(* Logix 5000 project; controller cal1632 1756-L62 rev 16.20; software revision 16.05; part 60 of 61 *)
(* tags used below, declared in another part *)
   A02 : ALIAS FOR hmi_dint[0].2;
   A08 : ALIAS FOR hmi_dint[0].8;
   A09 : ALIAS FOR hmi_dint[0].9;
   A10 : ALIAS FOR hmi_dint[0].10;
   A11 : ALIAS FOR hmi_dint[0].11;
   A12 : ALIAS FOR hmi_dint[0].12;
   A13 : ALIAS FOR hmi_dint[0].13;
   A14 : ALIAS FOR hmi_dint[0].14;
   A15 : ALIAS FOR hmi_dint[0].15;
   accum_filling_on : ALIAS FOR hmi_dint[9].12;
   accum_holding_pressure_on : BOOL;   // Accumulator Holding Pressure Active
   accum_tension_pressure_on : BOOL;   // Accumulator Tension Pressure Active
   accumulator_state : DINT;   // Accumulator Sequence State Word
   add_sys_Acknowledge : sys_Acknowledge;   // Addon Acknowledge
   add_sys_ramp : sys_Ramp;   // Addon Ramp
   ai_pos01_pct_flt : REAL;   // AI: Linear Position Transducer
   alarm_exists : ALIAS FOR hmi_dint[9].28;
   alm_ack : DINT[2];   // Accumulator Alarm Acknowledge Bits
   ao_prs01 : REAL;   // AO: Pressure 1
   ao_prs02 : REAL;   // AO: Pressure 2
   control_to_empty : ALIAS FOR hmi_dint[9].13;
   di_high_limit : ALIAS FOR p00_io_winder:6:I.0;
   di_ss_close_nip : ALIAS FOR p00_io_winder:5:I.14;
   di_ss_nip_auto : ALIAS FOR p00_io_winder:5:I.13;
   do_carriage_lift_sol : ALIAS FOR p00_io_winder:4:O.7;
   do_close_nip_sol : ALIAS FOR p00_io_winder:4:O.8;
   enable_control : BOOL;   // Accumulator - Enable Control
   filling_pressure : REAL;   // Accumulator Fill Pressure Tare + Tension + Fill PID Offset
   hmi_dint : DINT[20];
   lpt_raw_ok : BOOL;   // Accumulator LPT Raw Signal In Range
   Me : ALIAS FOR p00_wac;
   nip_close_request : ALIAS FOR hmi_dint[9].7;
   nip_mode_auto : BOOL;   // Nip Mode Auto
   nip_open_selected : BOOL;   // Nip Selector in OPEN Neither Auto nor Close
   param_acc_handover_band_pct : REAL;   // Parameter Accumulator Handover Band Stroke Over Which the Payout Boost Fades Out [% of Stroke]
   param_acc_handover_pct : REAL;
   param_acc_low_pstn_sp : REAL;   // Parameter Accumulator Low Position Setpoint
   param_acc_max_limit : REAL;   // Parameter Accumulator High Max Limit
   param_accel_rate : REAL;   // Parameter Acceleration Rate
   param_counter_prs : REAL;   // Parameter Counter Pressure
   param_cv01_manual_sp : REAL;
   param_decel_rate : REAL;   // Parameter Decleration Rate
   param_fill_SO : REAL;   // Parameter FIll Pressure
   param_gain : REAL;   // Parameter Gain
   param_high_ctrl_pct : REAL;   // Parameter High Control Position
   param_holding_pressure : REAL;   // Parameter Carriage Holding Pressure
   param_low_ctrl_pct : REAL;   // Parameter Low Control Position
   param_lpt_frozen_ms : DINT;   // Parameter LPT Frozen Detect Dwell [ms]
   param_pid_kp : REAL;   // Parameter PID Kp
   param_pid_process_type : DINT;   // PIDE Process Type Selected by Autotune at the HMI
   param_press_offset : REAL;   // Parameter Pressure Curve Offset Carriage weight term, vendor curve [lbf]
   param_press_slope_empty : REAL;   // Parameter Pressure Curve Slope - EMPTYING Web Tension lb = slope x psi - offset [lb/psi]
   param_press_slope_fill : REAL;   // Parameter Pressure Curve Slope - FILLING Web Tension lb = slope x psi - offset [lb/psi]
   param_tare_pressure : REAL;   // Parameter Friction Trim Pressure Carriage Balanced - No Drift Up or Down Set at Installation
   payout_active : BOOL;
   payout_pressure : REAL;
   pb_acc_on : ALIAS FOR hmi_dint[9].2;
   pb_enable_tension : ALIAS FOR local_pb.4;
   pb_reset : ALIAS FOR local_pb.31;
   pb_stop_line : ALIAS FOR local_pb.30;
   pid_ctrl_cv : REAL;   // PID Control CV
   pid_ctrl_pv : REAL;   // PID Control PV
   pid_ctrl_sp : REAL;   // PID Control SP
   pid_mode_manual : ALIAS FOR hmi_dint[9].15;
   PID_offset : REAL;   // Position PID Offset
   pstn_should_move : BOOL;   // Accumulator Position Must Be Changing Filling or Paying Out
   request_fill : ALIAS FOR hmi_dint[9].1;
   selected_pressure : REAL;   // Accumulator Selected Tension Pressure
   task_scan_time : REAL;   // Task Scan Time
   task_scan_time_dint : DINT;   // Task Scan
   tension_pressure : REAL;
   timer_alarm : TIMER[32];   // Accumulator Alarms Delay Timer
   timer_lpt_frozen : TIMER;   // Accumulator LPT Frozen Detect Timer
   timer_warning : TIMER[48];   // Accumulator Warning Delay
   unack_alarm : ALIAS FOR hmi_dint[9].29;
   unack_warning : ALIAS FOR hmi_dint[9].31;
   use_auto_tune_gains : BOOL;   // Tension PIDE Use Auto Tune Values
   W00 : ALIAS FOR hmi_dint[2].0;
   W01 : ALIAS FOR hmi_dint[2].1;
   W02 : ALIAS FOR hmi_dint[2].2;
   W03 : ALIAS FOR hmi_dint[2].3;
   W04 : ALIAS FOR hmi_dint[2].4;
   W05 : ALIAS FOR hmi_dint[2].5;
   W06 : ALIAS FOR hmi_dint[2].6;
   W07 : ALIAS FOR hmi_dint[2].7;
   wac_calc_tension_pressure : REAL;   // Winder Accumulator Calulated Tension Pressure
   wac_full_stop : BOOL;   // Accumulator Full - Normal Line Stop Requested Self-Clearing, No Reset Required
   wac_nearly_empty : BOOL;
   wac_tension_pressure : REAL;   // Winder Accumulator Tare + Web Tension Pressure Carriage Holds Position at Commanded Tension
   warning_exists : ALIAS FOR hmi_dint[9].30;
   winder_running : BOOL;   // Winder Running
   wrn_ack : DINT[2];   // Accumulator Warning Acknowledge Bits
   AFI : BOOL;
   FAULT : BOOL;
   HMI : BOOL;
   nip_mode_close : BOOL;   // Nip Mode Close
   p00_lin_timer_pre_0ms : DINT;
   p00_lin_timer_pre_1s : DINT;
   p00_lin_timer_pre_mcp : DINT;
   p00_lin_timer_pre_ms : DINT;
   p00_lin_timer_pre_ol : DINT;
   p00_wac : Accumulator;   // Winder Accumulator
   p00_wac_position_pct : REAL;   // Winder Accumulator Carriage Position Filtered [% of Stroke]
   p01_recipe_active : recipe;
   p01r09 : routine;
   p01r12_zero_line_speed : BOOL;
   p01r13_line_running : BOOL;
   p01r13_line_slow_ramp : BOOL;
   p29_winder_at_run_position : BOOL;
   p29r10 : routine;
   p29r11 : routine;
   p29r15_request_run : BOOL;
   p29r15_wdra_active : BOOL;
   p29r16_request_run : BOOL;
   p29r16_wdrb_active : BOOL;
(* P31_WAC, continued *)

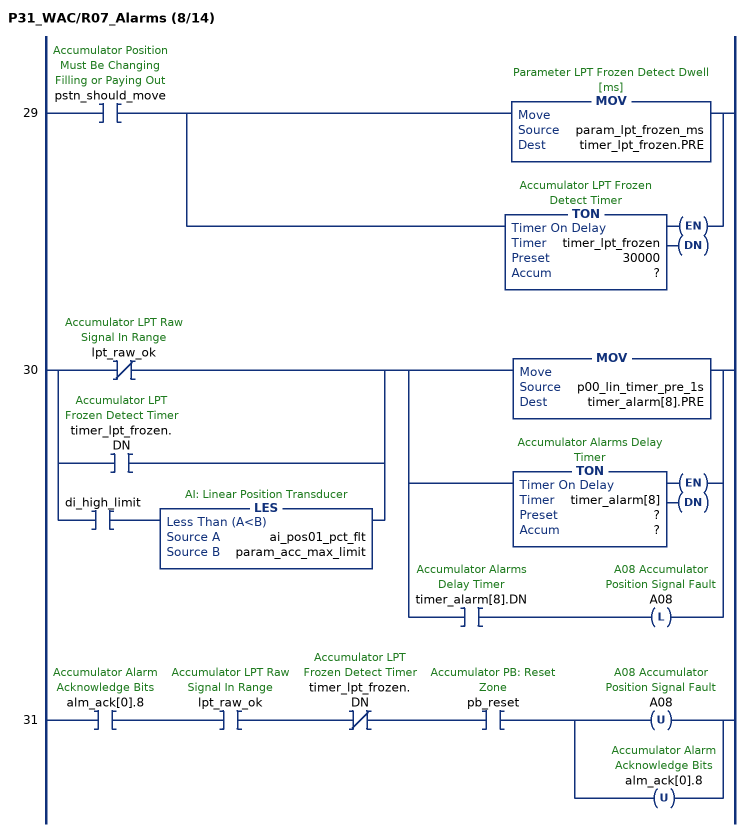
   [picture p1223: P31_WAC/R07_Alarms rungs 29-31]
   29: XIC(pstn_should_move)[MOV(param_lpt_frozen_ms,timer_lpt_frozen.PRE) ,TON(timer_lpt_frozen,?,?) ];
   30: [XIO(lpt_raw_ok) ,XIC(timer_lpt_frozen.DN) ,XIC(di_high_limit) LES(ai_pos01_pct_flt,param_acc_max_limit) ][MOV(p00_lin_timer_pre_1s,timer_alarm[8].PRE) ,TON(timer_alarm[8],?,?) ,XIC(timer_alarm[8].DN) OTL(A08) ];
   31: XIC(alm_ack[0].8)XIC(lpt_raw_ok)XIO(timer_lpt_frozen.DN)XIC(pb_reset)[OTU(A08) ,OTU(alm_ack[0].8) ];
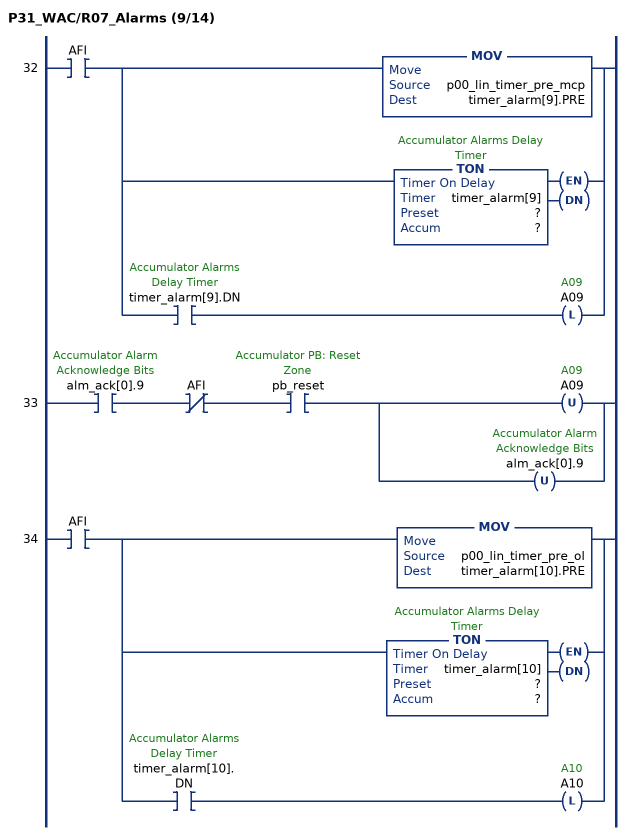
   32: XIC(AFI)[MOV(p00_lin_timer_pre_mcp,timer_alarm[9].PRE) ,TON(timer_alarm[9],?,?) ,XIC(timer_alarm[9].DN) OTL(A09) ];
   33: XIC(alm_ack[0].9)XIO(AFI)XIC(pb_reset)[OTU(A09) ,OTU(alm_ack[0].9) ];
   34: XIC(AFI)[MOV(p00_lin_timer_pre_ol,timer_alarm[10].PRE) ,TON(timer_alarm[10],?,?) ,XIC(timer_alarm[10].DN) OTL(A10) ];
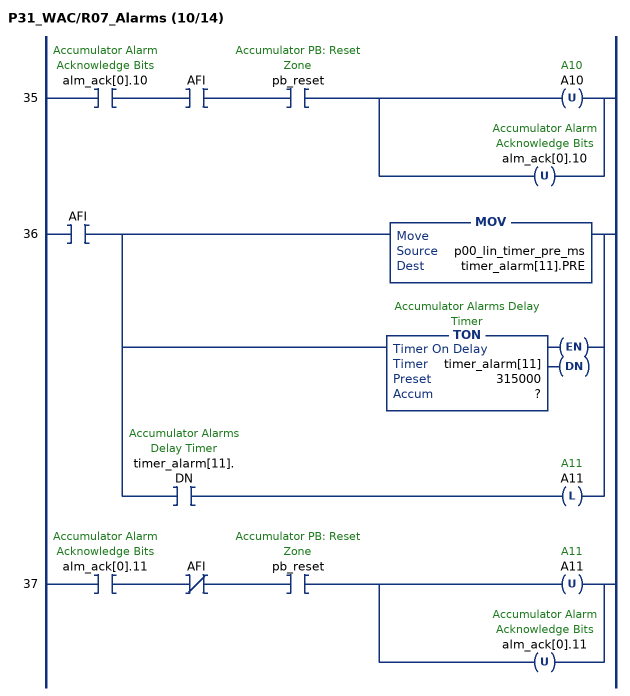
   35: XIC(alm_ack[0].10)XIC(AFI)XIC(pb_reset)[OTU(A10) ,OTU(alm_ack[0].10) ];
   36: XIC(AFI)[MOV(p00_lin_timer_pre_ms,timer_alarm[11].PRE) ,TON(timer_alarm[11],?,?) ,XIC(timer_alarm[11].DN) OTL(A11) ];
   37: XIC(alm_ack[0].11)XIO(AFI)XIC(pb_reset)[OTU(A11) ,OTU(alm_ack[0].11) ];
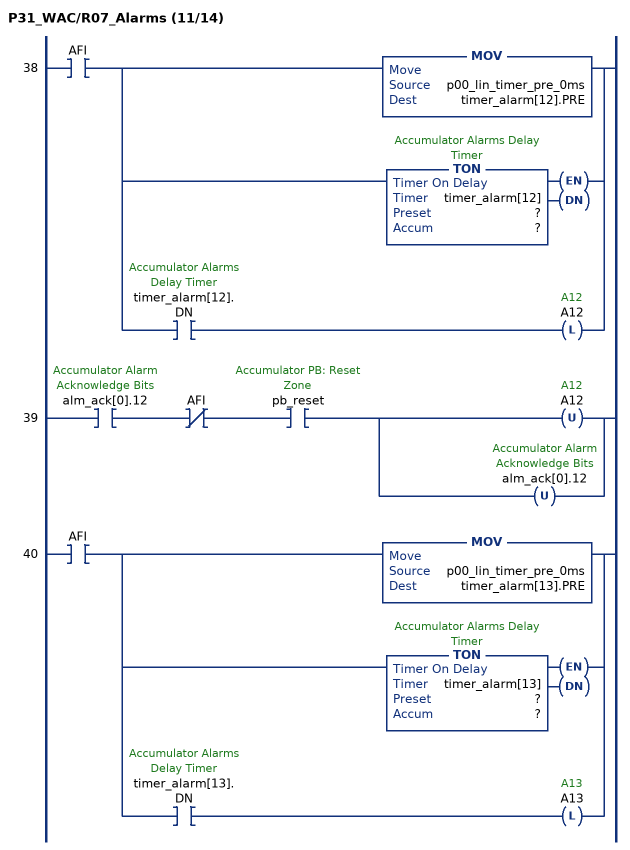
   38: XIC(AFI)[MOV(p00_lin_timer_pre_0ms,timer_alarm[12].PRE) ,TON(timer_alarm[12],?,?) ,XIC(timer_alarm[12].DN) OTL(A12) ];
   39: XIC(alm_ack[0].12)XIO(AFI)XIC(pb_reset)[OTU(A12) ,OTU(alm_ack[0].12) ];
   40: XIC(AFI)[MOV(p00_lin_timer_pre_0ms,timer_alarm[13].PRE) ,TON(timer_alarm[13],?,?) ,XIC(timer_alarm[13].DN) OTL(A13) ];
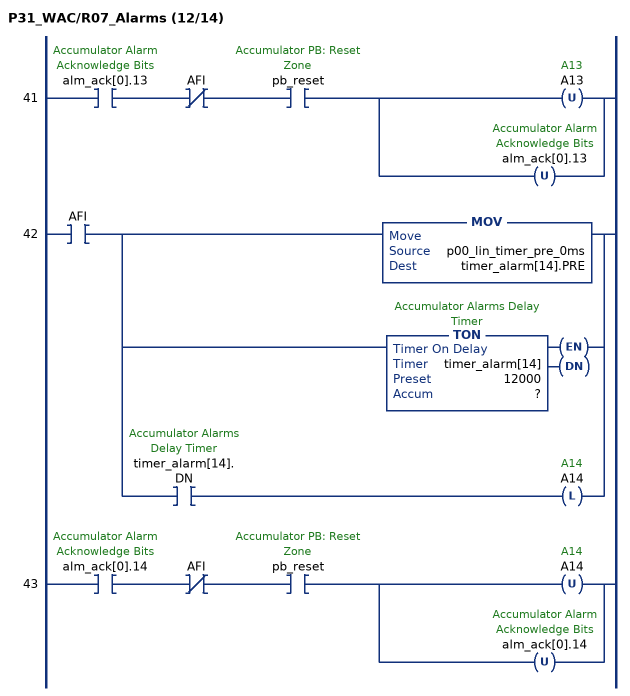
   41: XIC(alm_ack[0].13)XIO(AFI)XIC(pb_reset)[OTU(A13) ,OTU(alm_ack[0].13) ];
   42: XIC(AFI)[MOV(p00_lin_timer_pre_0ms,timer_alarm[14].PRE) ,TON(timer_alarm[14],?,?) ,XIC(timer_alarm[14].DN) OTL(A14) ];
   43: XIC(alm_ack[0].14)XIO(AFI)XIC(pb_reset)[OTU(A14) ,OTU(alm_ack[0].14) ];
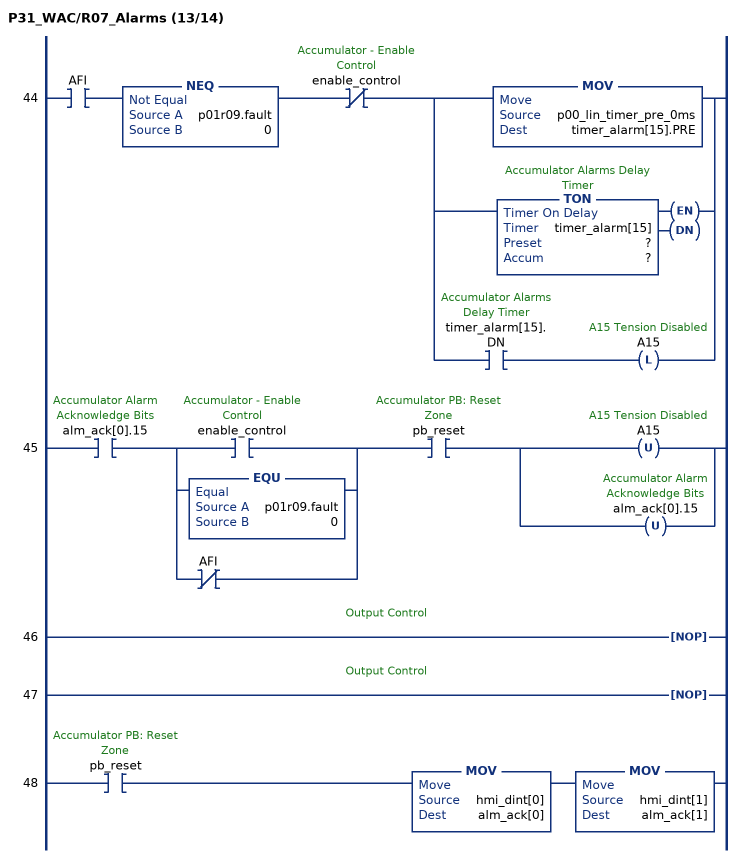
   44: XIC(AFI)NEQ(p01r09.fault,0)XIO(enable_control)[MOV(p00_lin_timer_pre_0ms,timer_alarm[15].PRE) ,TON(timer_alarm[15],?,?) ,XIC(timer_alarm[15].DN) OTL(A15) ];
   45: XIC(alm_ack[0].15)[[XIC(enable_control) ,EQU(p01r09.fault,0) ] ,XIO(AFI) ]XIC(pb_reset)[OTU(A15) ,OTU(alm_ack[0].15) ];
   // Output Control
   46: NOP();
   // Output Control
   47: NOP();
   48: XIC(pb_reset)MOV(hmi_dint[0],alm_ack[0])MOV(hmi_dint[1],alm_ack[1]);
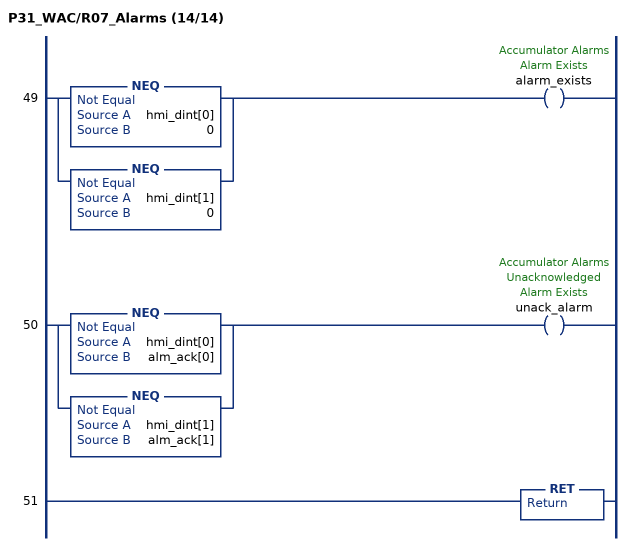
   49: [NEQ(hmi_dint[0],0) ,NEQ(hmi_dint[1],0) ]OTE(alarm_exists);
   50: [NEQ(hmi_dint[0],alm_ack[0]) ,NEQ(hmi_dint[1],alm_ack[1]) ]OTE(unack_alarm);
   51: RET();
END_ROUTINE

ROUTINE R08_Warnings   (* ladder *)
// Windup Accumulator
// Warnings
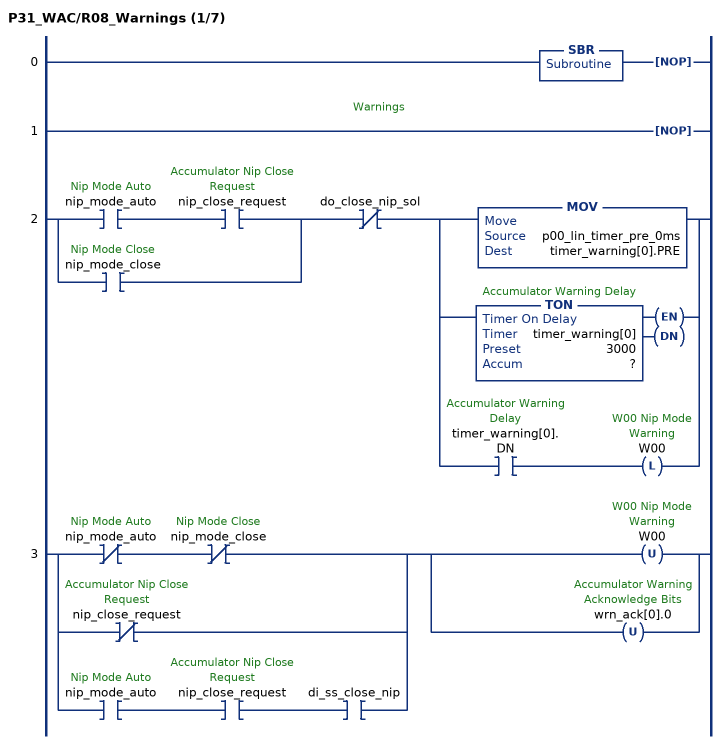
   0: SBR()NOP();
   // Warnings
   1: NOP();
   2: [XIC(nip_mode_auto) XIC(nip_close_request) ,XIC(nip_mode_close) ]XIO(do_close_nip_sol)[MOV(p00_lin_timer_pre_0ms,timer_warning[0].PRE) ,TON(timer_warning[0],?,?) ,XIC(timer_warning[0].DN) OTL(W00) ];
   3: [XIO(nip_mode_auto) XIO(nip_mode_close) ,XIO(nip_close_request) ,XIC(nip_mode_auto) XIC(nip_close_request) XIC(di_ss_close_nip) ][OTU(W00) ,OTU(wrn_ack[0].0) ];
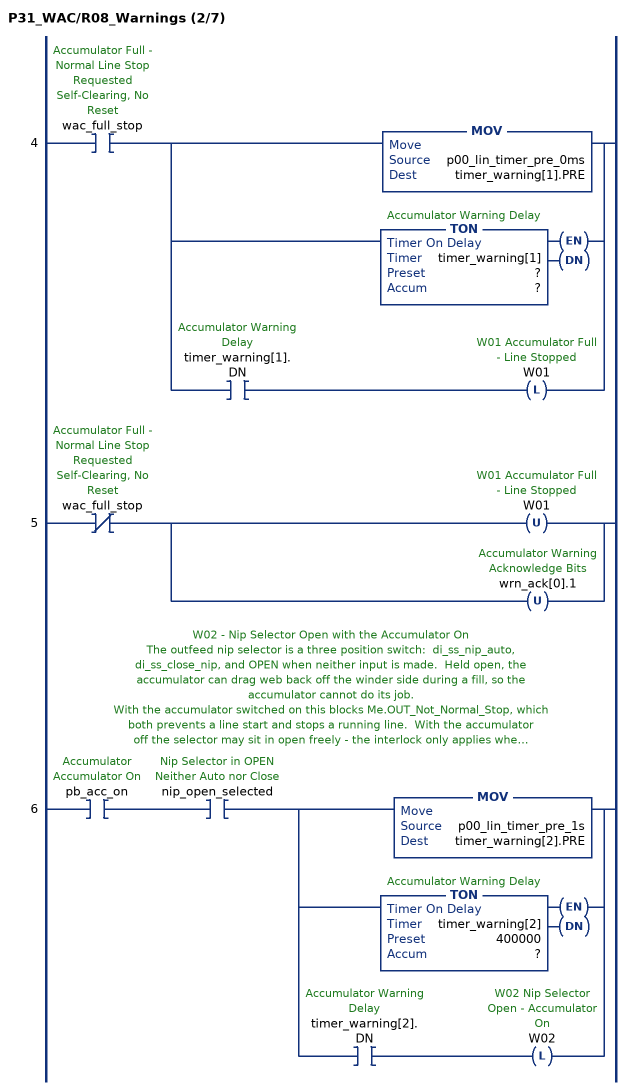
   4: XIC(wac_full_stop)[MOV(p00_lin_timer_pre_0ms,timer_warning[1].PRE) ,TON(timer_warning[1],?,?) ,XIC(timer_warning[1].DN) OTL(W01) ];
   5: XIO(wac_full_stop)[OTU(W01) ,OTU(wrn_ack[0].1) ];
   // W02 - Nip Selector Open with the Accumulator On
   // The outfeed nip selector is a three position switch:  di_ss_nip_auto,
   // di_ss_close_nip, and OPEN when neither input is made.  Held open, the
   // accumulator can drag web back off the winder side during a fill, so the
   // accumulator cannot do its job.
   // With the accumulator switched on this blocks Me.OUT_Not_Normal_Stop, which
   // both prevents a line start and stops a running line.  With the accumulator
   // off the selector may sit in open freely - the interlock only applies when
   // the accumulator is meant to be working.
   // This warning exists because the line simply refusing to start is not enough
   // for the operator to know why.  It clears itself as soon as either condition
   // goes away.
   // Rev 20260825 a12
   6: XIC(pb_acc_on)XIC(nip_open_selected)[MOV(p00_lin_timer_pre_1s,timer_warning[2].PRE) ,TON(timer_warning[2],?,?) ,XIC(timer_warning[2].DN) OTL(W02) ];
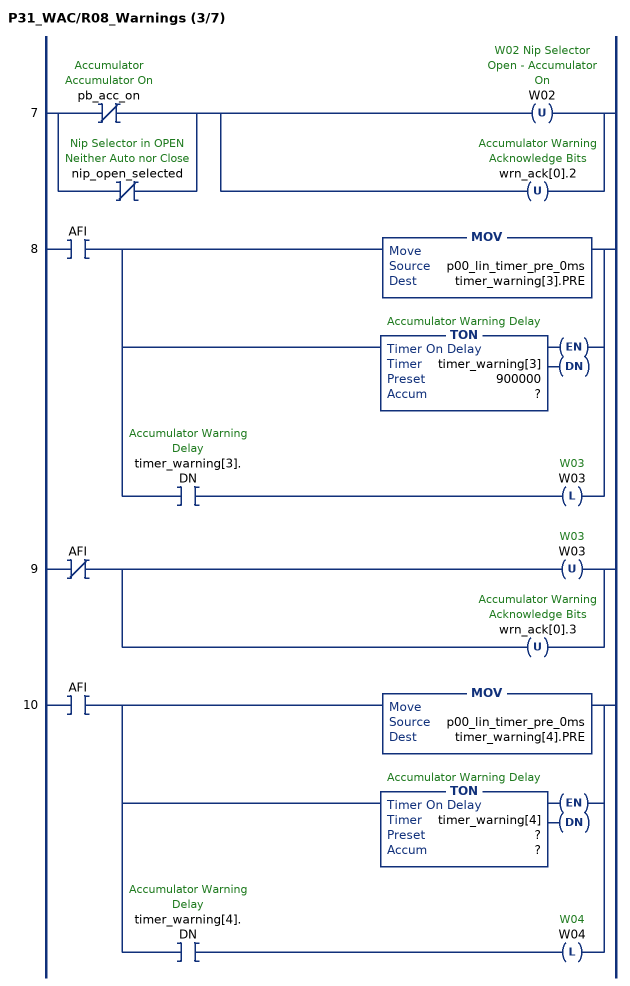
   7: [XIO(pb_acc_on) ,XIO(nip_open_selected) ][OTU(W02) ,OTU(wrn_ack[0].2) ];
   8: XIC(AFI)[MOV(p00_lin_timer_pre_0ms,timer_warning[3].PRE) ,TON(timer_warning[3],?,?) ,XIC(timer_warning[3].DN) OTL(W03) ];
   9: XIO(AFI)[OTU(W03) ,OTU(wrn_ack[0].3) ];
   10: XIC(AFI)[MOV(p00_lin_timer_pre_0ms,timer_warning[4].PRE) ,TON(timer_warning[4],?,?) ,XIC(timer_warning[4].DN) OTL(W04) ];
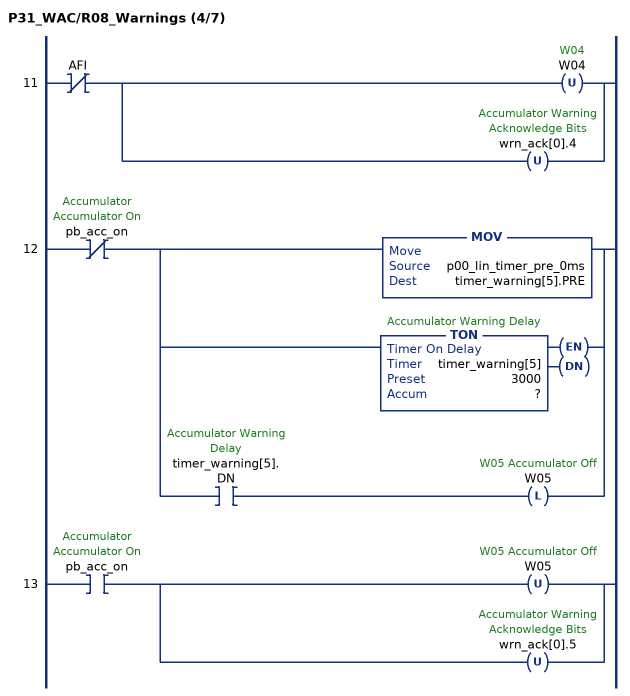
   11: XIO(AFI)[OTU(W04) ,OTU(wrn_ack[0].4) ];
   12: XIO(pb_acc_on)[MOV(p00_lin_timer_pre_0ms,timer_warning[5].PRE) ,TON(timer_warning[5],?,?) ,XIC(timer_warning[5].DN) OTL(W05) ];
   13: XIC(pb_acc_on)[OTU(W05) ,OTU(wrn_ack[0].5) ];
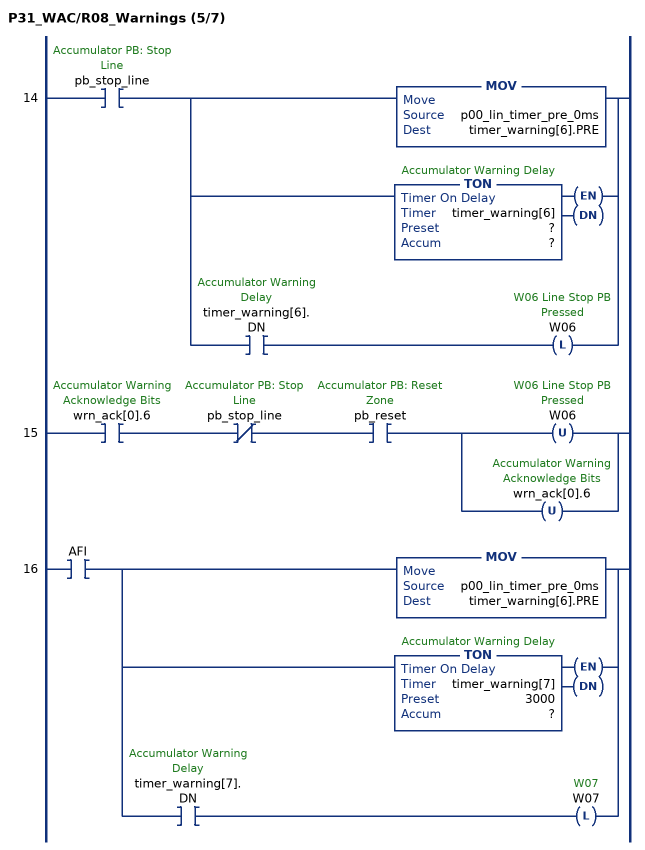
   14: XIC(pb_stop_line)[MOV(p00_lin_timer_pre_0ms,timer_warning[6].PRE) ,TON(timer_warning[6],?,?) ,XIC(timer_warning[6].DN) OTL(W06) ];
   15: XIC(wrn_ack[0].6)XIO(pb_stop_line)XIC(pb_reset)[OTU(W06) ,OTU(wrn_ack[0].6) ];
   16: XIC(AFI)[MOV(p00_lin_timer_pre_0ms,timer_warning[6].PRE) ,TON(timer_warning[7],?,?) ,XIC(timer_warning[7].DN) OTL(W07) ];
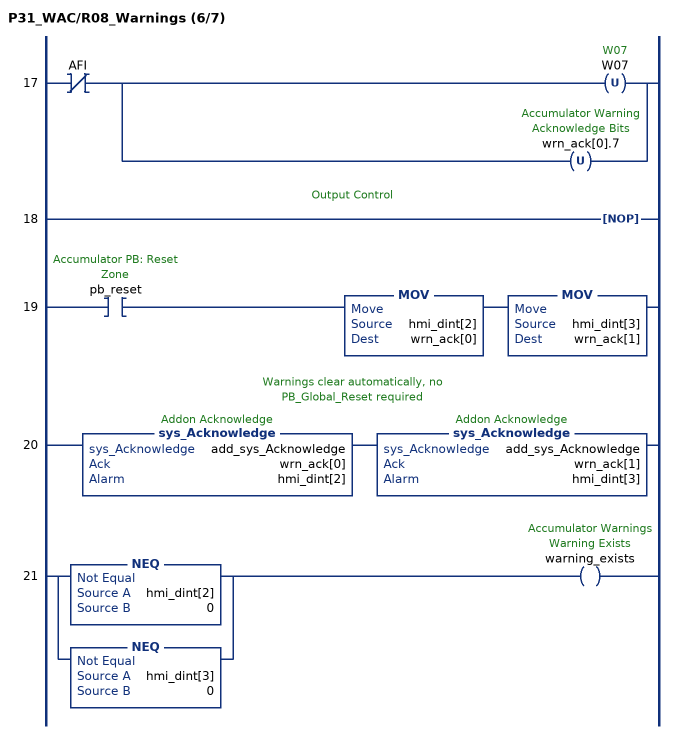
   17: XIO(AFI)[OTU(W07) ,OTU(wrn_ack[0].7) ];
   // Output Control
   18: NOP();
   19: XIC(pb_reset)MOV(hmi_dint[2],wrn_ack[0])MOV(hmi_dint[3],wrn_ack[1]);
   // Warnings clear automatically, no
   // PB_Global_Reset required
   20: sys_Acknowledge(add_sys_Acknowledge,wrn_ack[0],hmi_dint[2])sys_Acknowledge(add_sys_Acknowledge,wrn_ack[1],hmi_dint[3]);
   21: [NEQ(hmi_dint[2],0) ,NEQ(hmi_dint[3],0) ]OTE(warning_exists);
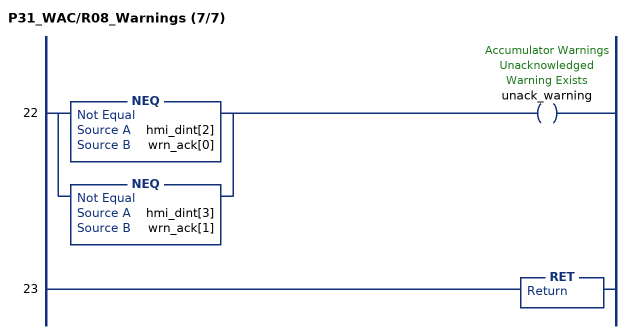
   22: [NEQ(hmi_dint[2],wrn_ack[0]) ,NEQ(hmi_dint[3],wrn_ack[1]) ]OTE(unack_warning);
   23: RET();
END_ROUTINE

ROUTINE R11_Modes   (* ladder *)
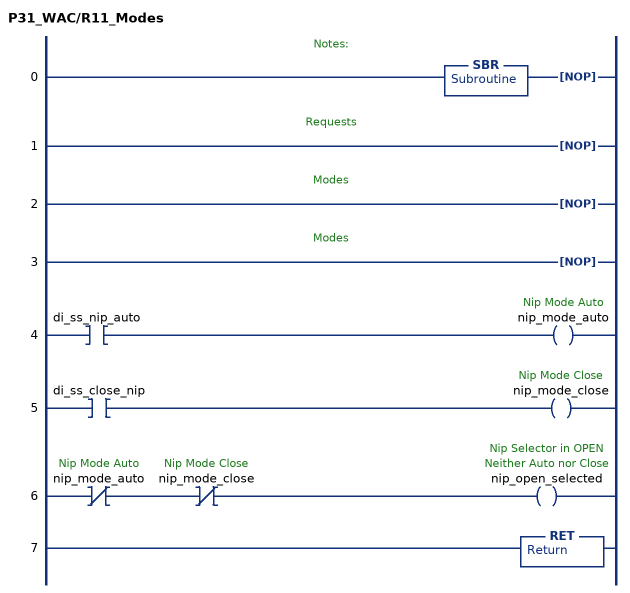
   // Notes:
   0: SBR()NOP();
   // Requests
   1: NOP();
   // Modes
   2: NOP();
   // Modes
   3: NOP();
   4: XIC(di_ss_nip_auto)OTE(nip_mode_auto);
   5: XIC(di_ss_close_nip)OTE(nip_mode_close);
   6: XIO(nip_mode_auto)XIO(nip_mode_close)OTE(nip_open_selected);
   7: RET();
END_ROUTINE

ROUTINE R21_Fill_Request   (* ladder *)
// WAC
// Fill Request and Tension Enable
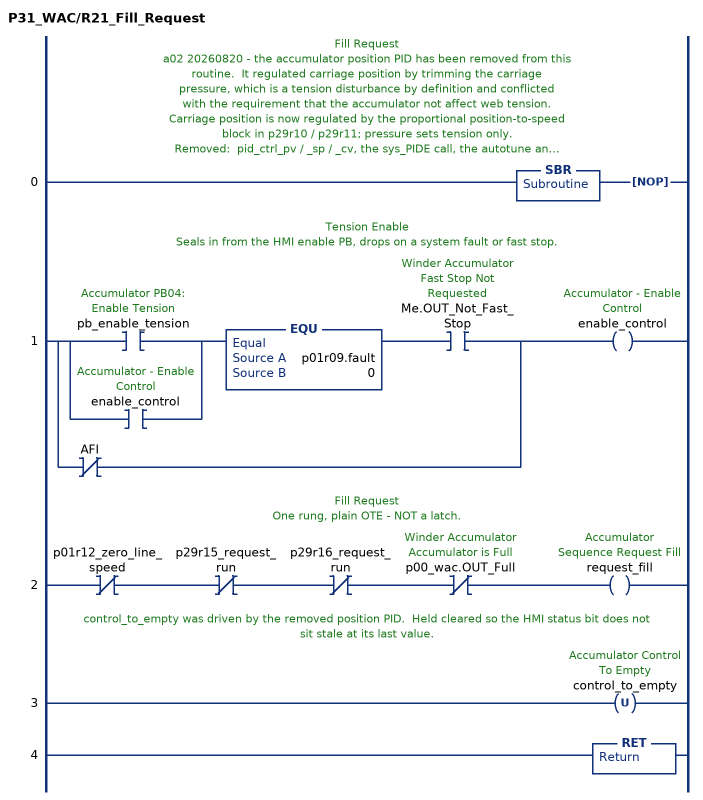
   // Fill Request
   // a02 20260820 - the accumulator position PID has been removed from this
   // routine.  It regulated carriage position by trimming the carriage
   // pressure, which is a tension disturbance by definition and conflicted
   // with the requirement that the accumulator not affect web tension.
   // Carriage position is now regulated by the proportional position-to-speed
   // block in p29r10 / p29r11; pressure sets tension only.
   // Removed:  pid_ctrl_pv / _sp / _cv, the sys_PIDE call, the autotune and
   //           gain plumbing, PIDE_ten manual mode and manual setpoint, and
   //           the PID_offset calculation.  The fill pressure bias that
   //           PID_offset used to supply now falls out of the separate
   //           vendor fill curve in p31 R22 - see param_press_slope_fill.
   // Kept declared for HMI back-compat, no longer consumed by any rung:
   //           PIDE_ten, PIDE_Control, pid_ctrl_pv, pid_ctrl_sp, pid_ctrl_cv,
   //           PID_offset, pid_mode_manual, use_auto_tune_gains, param_gain,
   //           param_pid_kp / ki / kd, param_pid_process_type, param_fill_SO,
   //           param_cv01_manual_sp, param_acc_low_pstn_sp,
   //           param_low_ctrl_pct, param_high_ctrl_pct.
   // What remains here is the fill request latch and the tension enable seal.
   // Routine renamed from R21_Position_PID; call order in R00_Main unchanged.
   0: SBR()NOP();
   // Tension Enable
   // Seals in from the HMI enable PB, drops on a system fault or fast stop.
   1: [[XIC(pb_enable_tension) ,XIC(enable_control) ] EQU(p01r09.fault,0) XIC(Me.OUT_Not_Fast_Stop) ,XIO(AFI) ]OTE(enable_control);
   // Fill Request
   // One rung, plain OTE - NOT a latch.
   2: XIO(p01r12_zero_line_speed)XIO(p29r15_request_run)XIO(p29r16_request_run)XIO(p00_wac.OUT_Full)OTE(request_fill);
   // control_to_empty was driven by the removed position PID.  Held cleared so the HMI status bit does not sit stale at its last value.
   3: OTU(control_to_empty);
   4: RET();
END_ROUTINE

ROUTINE R22_Fill_Pressure   (* ladder *)
// Windup Accumulator
// Fill Pressure
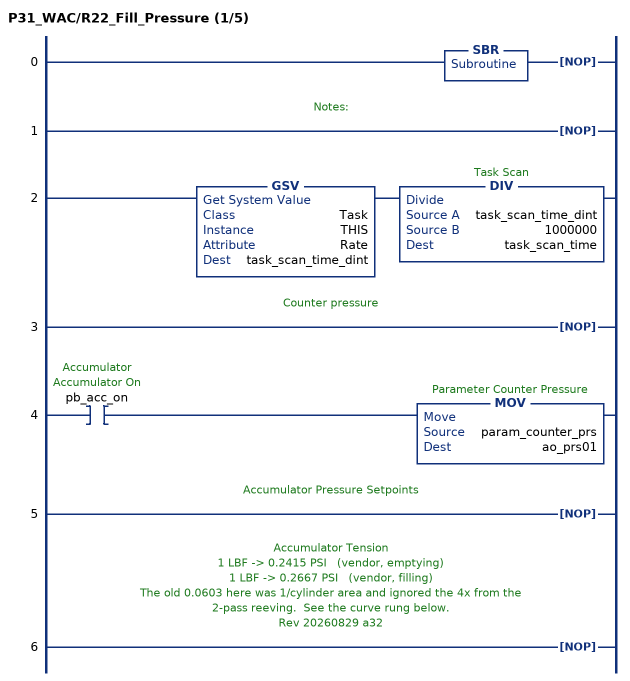
   0: SBR()NOP();
   // Notes:
   1: NOP();
   2: GSV(Task,THIS,Rate,task_scan_time_dint)DIV(task_scan_time_dint,1000000,task_scan_time);
   // Counter pressure
   3: NOP();
   4: XIC(pb_acc_on)MOV(param_counter_prs,ao_prs01);
   // Accumulator Pressure Setpoints
   5: NOP();
   // Accumulator Tension
   // 1 LBF -> 0.2415 PSI   (vendor, emptying)
   // 1 LBF -> 0.2667 PSI   (vendor, filling)
   // The old 0.0603 here was 1/cylinder area and ignored the 4x from the
   // 2-pass reeving.  See the curve rung below.
   // Rev 20260829 a32
   6: NOP();
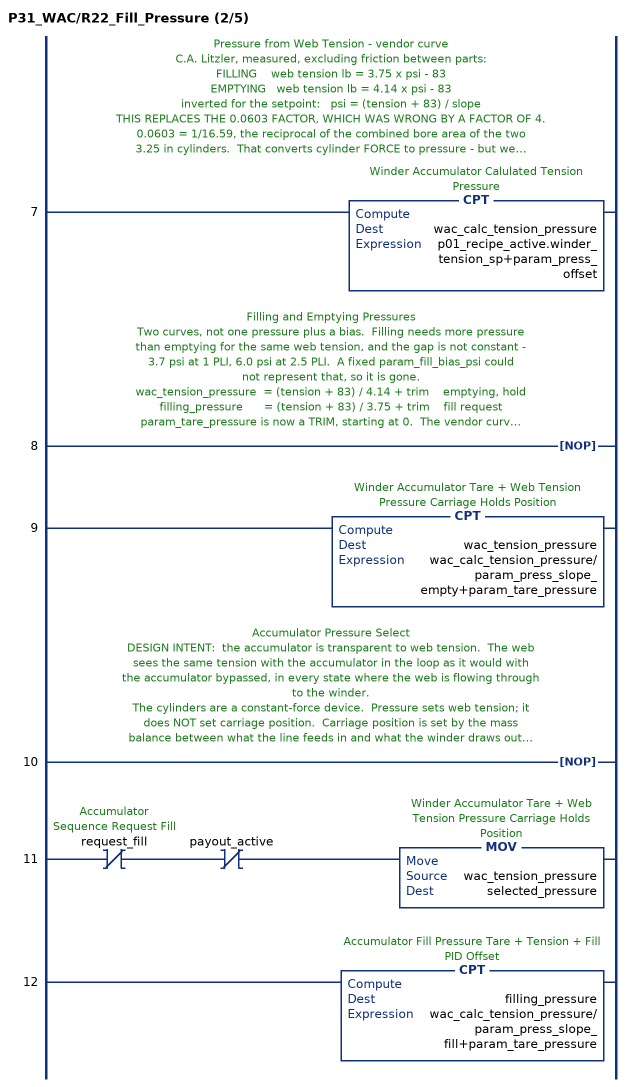
   // Pressure from Web Tension - vendor curve
   // C.A. Litzler, measured, excluding friction between parts:
   //   FILLING    web tension lb = 3.75 x psi - 83
   //   EMPTYING   web tension lb = 4.14 x psi - 83
   // inverted for the setpoint:   psi = (tension + 83) / slope
   // THIS REPLACES THE 0.0603 FACTOR, WHICH WAS WRONG BY A FACTOR OF 4.
   // 0.0603 = 1/16.59, the reciprocal of the combined bore area of the two
   // 3.25 in cylinders.  That converts cylinder FORCE to pressure - but web
   // tension is not cylinder force.  The carriage is reeved 2 passes, and
   // each pass puts two spans of web on the carriage, so the cylinders carry
   // 4 x T:
   //   psi = 4T/16.59 = 0.2411 T      vs vendor 1/4.14 = 0.2415 T
   // The old factor commanded a quarter of the pressure needed.  At 1 PLI the
   // tare masked it (34.6 vs 35.3 psi); at 2.5 PLI it was 40.3 psi against a
   // required 58.1 - the accumulator would have held about a third of the
   // tension asked for, and worse the higher the setpoint.
   // The 83 lbf offset is the carriage: 83 x 16.59/4 = 344 lb, consistent with
   // the mechanical note that the carriage must fall under its own weight.
   // Rev 20260829 a32
   7: CPT(wac_calc_tension_pressure,p01_recipe_active.winder_tension_sp+param_press_offset);
   // Filling and Emptying Pressures
   // Two curves, not one pressure plus a bias.  Filling needs more pressure
   // than emptying for the same web tension, and the gap is not constant -
   // 3.7 psi at 1 PLI, 6.0 psi at 2.5 PLI.  A fixed param_fill_bias_psi could
   // not represent that, so it is gone.
   //   wac_tension_pressure  = (tension + 83) / 4.14 + trim    emptying, hold
   //   filling_pressure      = (tension + 83) / 3.75 + trim    fill request
   // param_tare_pressure is now a TRIM, starting at 0.  The vendor curve
   // already carries the carriage weight in the 83 lbf offset, and is stated
   // to exclude friction between parts.  Any standing offset found at install
   // - seal drag, guide friction - goes here.  It is no longer the whole
   // intercept, so do NOT set it to 30.8.
   // Check against the vendor table at install:
   //   PLI   tension lb   fill psi   empty psi
   //   1.0        63        38.9       35.3
   //   1.5        94.5      47.3       42.9
   //   2.0       126        55.7       50.5
   //   2.5       157.5      64.1       58.1
   // Rev 20260829 a32
   8: NOP();
   9: CPT(wac_tension_pressure,wac_calc_tension_pressure/param_press_slope_empty+param_tare_pressure);
   // Accumulator Pressure Select
   // DESIGN INTENT:  the accumulator is transparent to web tension.  The web
   // sees the same tension with the accumulator in the loop as it would with
   // the accumulator bypassed, in every state where the web is flowing through
   // to the winder.
   // The cylinders are a constant-force device.  Pressure sets web tension; it
   // does NOT set carriage position.  Carriage position is set by the mass
   // balance between what the line feeds in and what the winder draws out.
   // Rungs are in order of increasing priority - the last rung to write
   // selected_pressure wins:
   //   1  Normal run                 wac_tension_pressure
   //   2  Payout                     wac_tension_pressure
   //   3  Fill request               filling_pressure  (steeper fill curve)
   //   4  Fault, or line not moving  wac_tension_pressure
   // 1, 2 and 4 are all the same pressure, and that is the point - nothing
   // about accumulator state changes web tension.  During payout the carriage
   // descends because the winder is overspeeding and drawing web out faster
   // than the line feeds it in, not because pressure was reduced.
   // The position PID offset is NO LONGER added to the running pressure.  Any
   // position trim on the pressure is a tension disturbance by definition, so
   // the carriage is left to float.  PID_offset now reaches the web only
   // through the fill bias in rung 3, where the exit nip is closed and the
   // winder is isolated from the accumulator.
   // Superseded, no longer used:  payout_pressure (fixed 29 psi),
   // param_holding_pressure (fixed 14 psi), tension_pressure (fixed 35 psi).
   // Rev 20260820
   10: NOP();
   11: XIO(request_fill)XIO(payout_active)MOV(wac_tension_pressure,selected_pressure);
   12: CPT(filling_pressure,wac_calc_tension_pressure/param_press_slope_fill+param_tare_pressure);
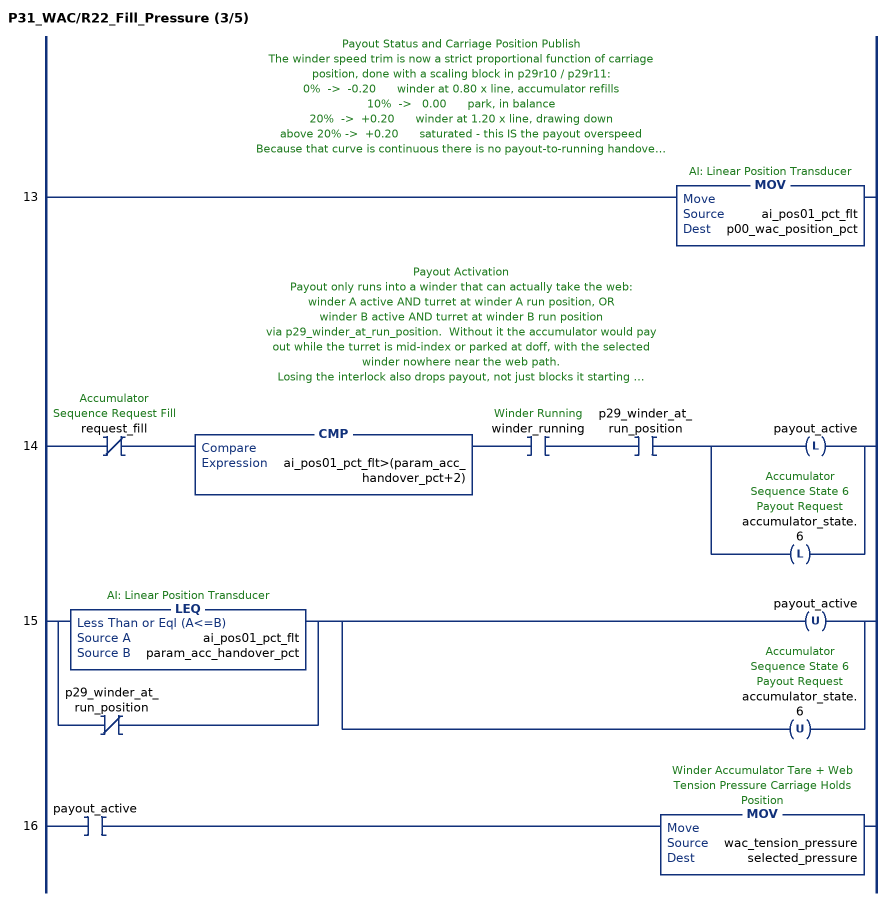
   // Payout Status and Carriage Position Publish
   // The winder speed trim is now a strict proportional function of carriage
   // position, done with a scaling block in p29r10 / p29r11:
   //         0%  ->  -0.20      winder at 0.80 x line, accumulator refills
   //        10%  ->   0.00      park, in balance
   //        20%  ->  +0.20      winder at 1.20 x line, drawing down
   //    above 20% ->  +0.20      saturated - this IS the payout overspeed
   // Because that curve is continuous there is no payout-to-running handover
   // to sequence and no cross-fade.  The accumulator seeks 10% on its own,
   // which also removes the position drift that a purely tension-transparent
   // accumulator would otherwise show over a long run.
   // p00_wac_position_pct is the filtered carriage position published to p29.
   // P31 scans after P29 so p29 reads it one scan old - 10 ms on a carriage
   // that moves slowly, which is not significant.
   // payout_active / accumulator_state.6 / Me.OUT_Acc_Payout are retained as
   // STATUS ONLY - HMI indication and the pressure select rungs below.  They
   // no longer gate any speed logic.  Latch is at park + 2% so that a short
   // doff which only part-fills still shows payout; unlatch at park, with
   // wac_nearly_empty kept as a backstop.
   // Rev 20260820
   13: MOV(ai_pos01_pct_flt,p00_wac_position_pct);
   // Payout Activation
   // Payout only runs into a winder that can actually take the web:
   //   winder A active AND turret at winder A run position, OR
   //   winder B active AND turret at winder B run position
   // via p29_winder_at_run_position.  Without it the accumulator would pay
   // out while the turret is mid-index or parked at doff, with the selected
   // winder nowhere near the web path.
   // Losing the interlock also drops payout, not just blocks it starting -
   // the turret can be jogged away underneath an active payout.
   // Rev 20260829 a33
   14: XIO(request_fill)CMP(ai_pos01_pct_flt>(param_acc_handover_pct+2))XIC(winder_running)XIC(p29_winder_at_run_position)[OTL(payout_active) ,OTL(accumulator_state.6) ];
   15: [LEQ(ai_pos01_pct_flt,param_acc_handover_pct) ,XIO(p29_winder_at_run_position) ][OTU(payout_active) ,OTU(accumulator_state.6) ];
   16: XIC(payout_active)MOV(wac_tension_pressure,selected_pressure);
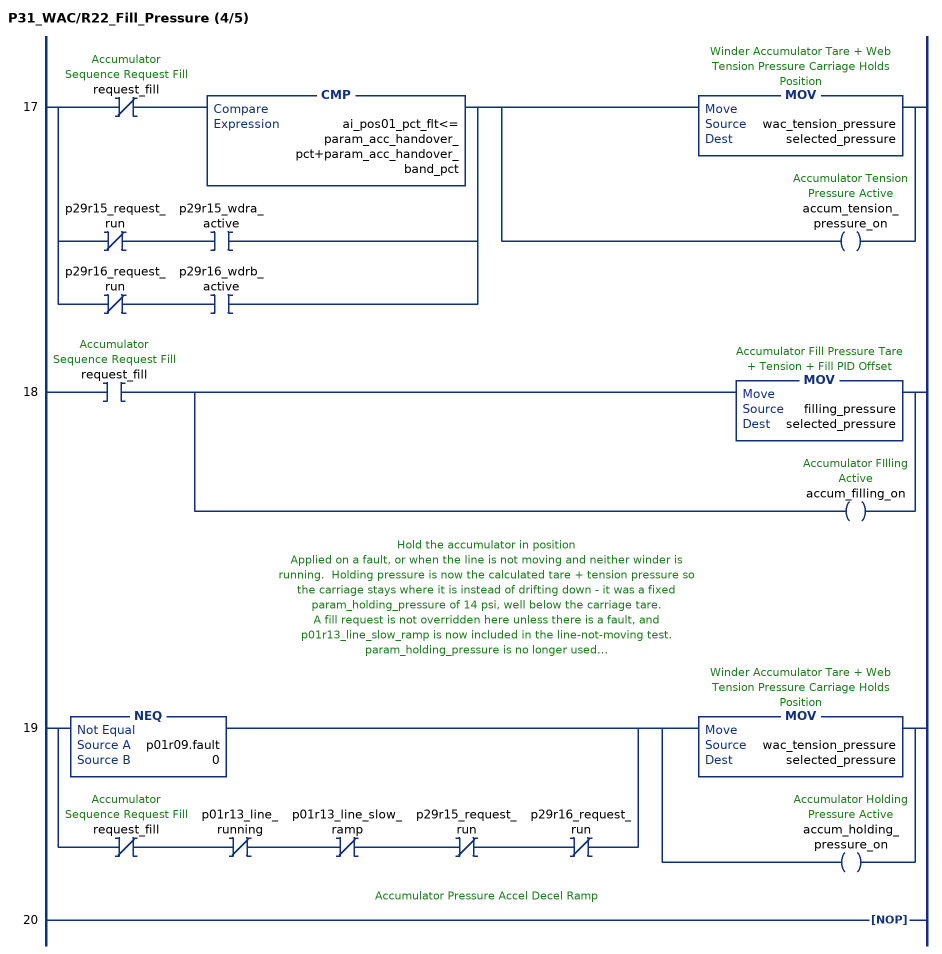
   17: [XIO(request_fill) CMP(ai_pos01_pct_flt<= param_acc_handover_pct+param_acc_handover_band_pct) ,XIO(p29r15_request_run) XIC(p29r15_wdra_active) ,XIO(p29r16_request_run) XIC(p29r16_wdrb_active) ][MOV(wac_tension_pressure,selected_pressure) ,OTE(accum_tension_pressure_on) ];
   18: XIC(request_fill)[MOV(filling_pressure,selected_pressure) ,OTE(accum_filling_on) ];
   // Hold the accumulator in position
   // Applied on a fault, or when the line is not moving and neither winder is
   // running.  Holding pressure is now the calculated tare + tension pressure so
   // the carriage stays where it is instead of drifting down - it was a fixed
   // param_holding_pressure of 14 psi, well below the carriage tare.
   // A fill request is not overridden here unless there is a fault, and
   // p01r13_line_slow_ramp is now included in the line-not-moving test.
   // param_holding_pressure is no longer used.
   // Rev 20260820
   19: [NEQ(p01r09.fault,0) ,XIO(request_fill) XIO(p01r13_line_running) XIO(p01r13_line_slow_ramp) XIO(p29r15_request_run) XIO(p29r16_request_run) ][MOV(wac_tension_pressure,selected_pressure) ,OTE(accum_holding_pressure_on) ];
   // Accumulator Pressure Accel Decel Ramp
   20: NOP();
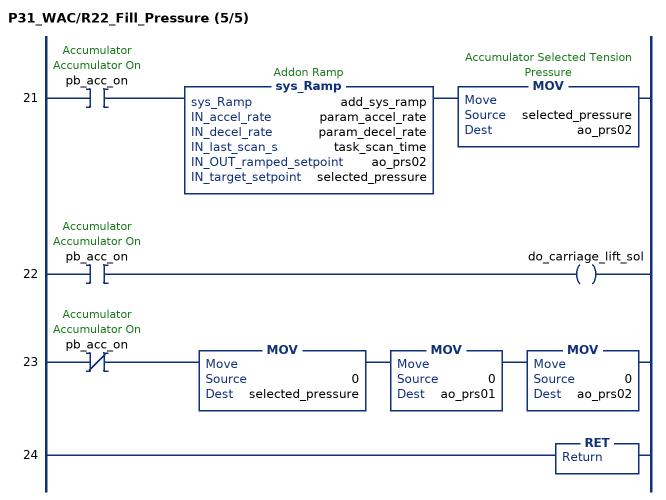
   21: XIC(pb_acc_on)sys_Ramp(add_sys_ramp,param_accel_rate,param_decel_rate,task_scan_time,ao_prs02,selected_pressure)MOV(selected_pressure,ao_prs02);
   22: XIC(pb_acc_on)OTE(do_carriage_lift_sol);
   23: XIO(pb_acc_on)MOV(0,selected_pressure)MOV(0,ao_prs01)MOV(0,ao_prs02);
   24: RET();
END_ROUTINE
